// TIA Portal V20 export
TYPE "typeSafetyDriveStatus"
// Safety status of drive
// stored: Access Published, IsFailsafeCompliant true, Namespace Safety
   STRUCT
      drive1 { S7_SetPoint := 'True'} : "Safety.typeSafetyDrive";
      drive2 { S7_SetPoint := 'True'} : "Safety.typeSafetyDrive";
      drive3 { S7_SetPoint := 'True'} : "Safety.typeSafetyDrive";
      drive4 { S7_SetPoint := 'True'} : "Safety.typeSafetyDrive";
      drive5 { S7_SetPoint := 'True'} : "Safety.typeSafetyDrive";
      drive6 { S7_SetPoint := 'True'} : "Safety.typeSafetyDrive";
      drive7 { S7_SetPoint := 'True'} : "Safety.typeSafetyDrive";
      drive8 { S7_SetPoint := 'True'} : "Safety.typeSafetyDrive";
      drive9 { S7_SetPoint := 'True'} : "Safety.typeSafetyDrive";
      drive10 { S7_SetPoint := 'True'} : "Safety.typeSafetyDrive";
      drive11 { S7_SetPoint := 'True'} : "Safety.typeSafetyDrive";
      drive12 { S7_SetPoint := 'True'} : "Safety.typeSafetyDrive";
      drive13 { S7_SetPoint := 'True'} : "Safety.typeSafetyDrive";
      drive14 { S7_SetPoint := 'True'} : "Safety.typeSafetyDrive";
      drive15 { S7_SetPoint := 'True'} : "Safety.typeSafetyDrive";
      drive16 { S7_SetPoint := 'True'} : "Safety.typeSafetyDrive";
      drive17 { S7_SetPoint := 'True'} : "Safety.typeSafetyDrive";
      drive18 { S7_SetPoint := 'True'} : "Safety.typeSafetyDrive";
   END_STRUCT;
END_TYPE
